FUNCTION CoolTank
VAR_INPUT
	refIn : REFERENCE TO ST_Tank;
END_VAR
VAR
	rSafeTemp : REAL := 50;
END_VAR

IF refIn.rtemperature >80 THEN
      refIn.rtemperature := refIn.rtemperature - 1;
END_IF

END_FUNCTION

(* stored: Version 1.1.0.1, ProductVersion 3.1.4024.16
   POU CoolTank: Id {2cc98c59-0933-4d64-9a53-53333cea12b3}, SpecialFunc None *)
